// TIA Portal V17 export
// export: Created 2025-06-25T13:13:27.972094Z, ExportSetting WithDefaults, DisplayName Totally Integrated Automation Portal, DisplayVersion V17 Update 8, DisplayName TIA Portal Openness, DisplayVersion V17 Update 8, DisplayName TIA Portal Version Control Interface, DisplayVersion V17, DisplayName STEP 7 Professional, DisplayVersion V17 Update 8, DisplayName STEP 7 Safety, DisplayVersion V17 Update 6, DisplayName WinCC Advanced, DisplayVersion V17 Update 8
TYPE "stABB_ACSx80_Rx"
// stored: IsFailsafeCompliant false
   STRUCT
      SW : Word;   // Status Word (58.109)
      Act1 : Word;   // Actual value 1 (58.110)
      Act2 : Word;   // Actual value 2 (58.111)
      DataIO_12 : Word;   // User configurable 1 (58.112)
      DataIO_13 : Word;   // User configurable 2 (58.113)
      DataIO_14 : Word;   // User configurable 3 (58.114)
      DataIO_15 : Word;   // User configurable 4 (58.115)
      DataIO_16 : Word;   // User configurable 5 (58.116)
   END_STRUCT;
END_TYPE
